Staubli VAL3: page_home_set.pjx

--- page_home_set.pjx ---
Parameters version=s7.6.3 stackSize=5000 millimeterUnit=true
Program file=alreadyExist.pgx
Program file=buildList.pgx
Program file=dataListAdd.pgx
Program file=deleteItem.pgx
Program file=listAdd.pgx
Program file=loadPage.pgx
Program file=main.pgx
Program file=markListAdd.pgx
Program file=markTraj.pgx
Program file=onEnterEvent.pgx
Program file=onExit.pgx
Program file=onF1Event.pgx
Program file=onF2Event.pgx
Program file=onF3Event.pgx
Program file=onF4Event.pgx
Program file=onF5Event.pgx
Program file=onF6Event.pgx
Program file=onF7Event.pgx
Program file=onF8Event.pgx
Program file=onLeftEvent.pgx
Program file=onRightEvent.pgx
Program file=onStart.pgx
Program file=refresh.pgx
Program file=refreshDynamic.pgx
Program file=refreshStatic.pgx
Program file=Wizard_bigBox.pgx
Program file=Wizard_smlBox.pgx
Data file=page_home_set.dtx
Library alias=page path=Disk://kernel/template/page/page.pjx
Library alias=use path=Disk://goHome/userPage/userPage.pjx
Library alias=home path=Disk://goHome/goHome.pjx
Library alias=save path=Disk://goHome/saveHomeBox/saveHomeBox.pjx
Library alias=set path=Disk://goHome/goHome.pjx
Library alias=language2 path=Disk://goHome/language/language.pjx
Library alias=cycleStatus path=Disk://cycleStatus/cycleStatus.pjx
Library alias=saveData path=Disk://saveData/saveData.pjx
Library alias=language path=Disk://kernel/language/language.pjx
Library alias=TRAJ path=Disk://trajectory/TRAJ/TRAJ.pjx
Library alias=JPOINT path=Disk://trajectory/JPOINT/JPOINT.pjx

--- page_home_set.dtx ---
public string sItems
num nKey
num nIndex
public string sEvent
num nView
num nSelected
string sList
public string sMenuUser[8]
num nRefresh
num nTime = 0.5
string sMenu
bool bLarge
bool bButton[8]
num nInsert
string sMarkList
string sDataList
num nSelected1

--- main.pgx ---
public program main()
  local num i
  local bool l_bSave
  local string sButton[3]
  local string sItems[2]
begin
  call onStart()
  do
    call refresh()
    nKey=getKey()
    call use:listevent(nKey,nIndex,sEvent)
    nView=use:nView
    nSelected=nIndex
    //
    // OVERRIDE NORMAL FUNCTIONALITY-> POLYMORPHISM
    //
    switch nKey
      case 264
        // left
        call onLeftEvent()
      break
      case 268
        // right
        call onRightEvent()
      break
      case 271
        // test
        call onF1Event()
      break
      case 272
        //
        call onF2Event()
      break
      case 273
        call onF3Event()
      break
      case 274
        call onF4Event()
      break
      case 275
        //
        call onF5Event()
      break
      case 276
        // set type
        call onF6Event()
      break
      case 277
        // DELETE
        call onF7Event()
      break
      case 278
        // NEW
        call onF8Event()
        l_bSave=true
      break
      case 270
        call onEnterEvent()
      break
    endSwitch
    // release the resource
    delay(0)
  until nKey==255 and isKeyPressed(289)==false
  // exit
  call onExit(l_bSave)
end

--- alreadyExist.pgx ---
program alreadyExist(string& x_sName[], bool& x_bUndo[])
  local num l_nX
  local num l_nY
  local string l_sString
begin
  // look if the trajectory already exist
  l_nX=40-use:nBottomX-1
  l_nY=use:nBottomY+1
  call language:message(l_sString,21)
  call use:type(l_nX,l_nY,l_sString)
  // read the new trajectory
  call use:read(l_nX+len(l_sString),l_nY,x_sName,10,false)
  if !use:bUseEscape
    call set:find(x_sName,x_bUndo)
    if x_bUndo
      call language:message(x_sName,-2)
      popUpMsg(x_sName)
    endIf
  else
    x_bUndo=true
  endIf
end

--- buildList.pgx ---
program buildList()
  local num i
  local bool l_bFound
  local num l_nCount
  local num l_nSize
  local string l_sEmpty
  local string l_sEvent
begin
  // INIT the list
  l_sEmpty=""
  call use:stringCopy(l_sEmpty,sList)
  // Build the list
  call home:getBoxSize(save:nBoxType,l_nSize)
  for i=0 to l_nSize-1
    call set:getEvent(l_sEvent,i,save:nBoxType)
    if l_sEvent!=""
      //
      // use the filter ?
      //
      // check if the bProcessList filter is active
      //
      l_bFound=true
      // update the selected item
      if l_sEvent==sEvent
        nSelected=l_nCount
      endIf
      // add
      if l_bFound
        call listAdd(l_sEvent)
        l_nCount=l_nCount+1
      endIf
    endIf
  endFor
  // update
  use:bUseRefresh=true
end

--- dataListAdd.pgx ---
program dataListAdd(string x_sEvent)
begin
  // add in the queue
  if sDataList!=""
    insert(sDataList[size(sDataList)])
  endIf
  sDataList[size(sDataList)-1]=x_sEvent
end

--- deleteItem.pgx ---
program deleteItem(bool& x_bResult)
  local string l_sMessage
  local string l_sButton[2]
  local string l_sTitle
  local bool l_bYes
begin
  x_bResult=false
  //delete it
  call language2:message(l_sMessage,3)
  call language:getYesNo(l_sButton)
  call set:getListTitle(l_sTitle)
  call use:yes_no(l_sMessage+"#"+l_sTitle+" "+sEvent,l_sButton,l_bYes)
  x_bResult=l_bYes
end

--- loadPage.pgx ---
program loadPage(string x_sPage (dimensions=1), string& x_sItems[] (dimensions=1))
// load the next page
  local num i
begin
  // look if the page libload is correct
  i=page:libLoad(x_sPage)
  if i!=0
    logMsg("[VALPLAST] INTERFACE:PAGE LIBLOAD "+x_sPage+" result "+toString("",i))
    popUpMsg("Loading page "+x_sPage+" error CODE "+toString("",i))
  else
    // copy all the field from x_sItems to the next page
    page:sItems=x_sItems
    call page:main()
    // to give back
    x_sItems=page:sItems
  endIf
end

--- markListAdd.pgx ---
program markListAdd(string x_sEvent)
begin
  // add in the queue
  if sMarkList!=""
    insert(sMarkList[size(sMarkList)])
  endIf
  sMarkList[size(sMarkList)-1]=x_sEvent
end

--- markTraj.pgx ---
program markTraj(num& x_nResult)
  local string l_sMessage[2]
  local num l_nTRAJ
  local num l_nJPOINT
  local string l_sKey
  local num i
  local string l_sItem
  local bool l_bRefresh
  local string l_sEmpty
  local num l_nView
  local string l_sEvent
  local bool l_bFound
  local num l_nCount
  local bool l_bSelected
  local num l_nSelected
  local bool l_bOk
begin
  //********************get data list*********//
  call use:stringCopy(l_sEmpty,sDataList)
  call TRAJ:getSize(l_nTRAJ)
  call JPOINT:getSize(l_nJPOINT)
  for i=0 to l_nTRAJ-1
    call TRAJ:get(l_sKey,i)
    l_sMessage="TRAJ "+l_sKey
    call dataListAdd(l_sMessage)
  endFor
  for i=0 to l_nJPOINT-1
    call JPOINT:get(l_sKey,i)
    l_sMessage="JPOINT "+l_sKey
    call dataListAdd(l_sMessage)
  endFor
  l_bRefresh=true
  do
    //******************************************//
    //******************bulid list*****************//
    for i=0 to size(sDataList)-1
      l_sEvent=sDataList[i]
      if l_sEvent!=""
        l_bFound=true
        // update the selected item
        if l_sEvent==sEvent
          nSelected=l_nCount
        endIf
        // add
        if l_bFound
          l_nCount=l_nCount+1
        endIf
      endIf
    endFor
    do

      if l_bRefresh==true
        l_bRefresh=false
        cls()
        // define your list size for default
        call use:setSizeList(0,0,22,11)
        call use:setView(false)
        call use:listcreate("")
        call use:listadd(sDataList)
        call use:clear(0,13)
        call language2:message(l_sMessage,5)
        call use:type(1,13,l_sMessage)
        call use:type(32,13,"#")
        call use:type(37,13,"OK")
        // refresh the list
        call use:selectNewField(nSelected,nIndex,nView)
        call refreshDynamic()
      else
        // refresh the Dynamic message
        if abs(clock()-nRefresh)>nTime
          call refreshDynamic()
        endIf
      endIf
      nKey=getKey()
      call use:listevent(nKey,nIndex,sEvent)
      nView=use:nView
      nSelected=nIndex
      switch nKey
        case 277
          if sEvent !=""
            if left(sDataList[nIndex],1)!="#"
              sDataList[nIndex]="# "+sDataList[nIndex]
              l_bRefresh=true
            else
              sDataList[nIndex]=right(sDataList[nIndex],len(sDataList[nIndex])-2)
              l_bRefresh=true
            endIf
          endIf
          call use:nullKey(nKey)
        break
        case 278
          l_bSelected=true
          call use:nullKey(nKey)
        break
      endSwitch
      delay(0)
    until nKey==255  or l_bRefresh==true or l_bSelected==true
    if l_bSelected==true
      //**********************已经选择的部分**********************//
      call use:stringCopy(l_sEmpty,sMarkList)
      do
        l_bRefresh=false
        cls()
        // create the list
        call use:setSizeList(12,0,25,11)
        call use:clear(0,13)
        call language2:message(l_sMessage,8)
        call use:type(31,13,l_sMessage)
        call language2:message(l_sMessage,7)
        call use:type(36,13,l_sMessage)
        // get the value

        //add mark list
        for i=0 to size(sDataList)-1
          if left(sDataList[i],1)=="#"
            call markListAdd(right(sDataList[i],len(sDataList[i])-2))
          endIf
        endFor
        if sMarkList==""
          l_nSelected=0
        else
          l_nSelected=size(sMarkList)
        endIf
        call language2:message(l_sMessage[0],52)
        call language2:message(l_sMessage[1],53)

        call use:listcreate(l_sMessage[0]+toString("",l_nSelected)+l_sMessage[1])
        //
        for i=0 to size(sMarkList)-1
          l_sItem=sMarkList[i]
          call use:listadd(l_sItem)
        endFor

        //////////bulid list
        ////////////////////
        // list update
        call use:listupdate(min(nInsert,size(sMarkList)))

        // Select ???
        do
          nKey=get()
          call use:listevent(nKey,nInsert,l_sItem)
          // release the resource
          if nKey==277
            l_bRefresh=true
            l_bSelected=false
            call use:nullKey(nKey)
          endIf
          if nKey==278
            if sMarkList==""
              call language2:message(l_sMessage,9)
              popUpMsg(l_sMessage)
              cls()
              use:bUseRefresh=true
              wait(getKey( )==-1)
              x_nResult=-1
              return
            endIf
            call set:IsUseSameTool(sMarkList,l_bOk)
            if l_bOk==false
              call language2:message(l_sMessage,54)
              popUpMsg(l_sMessage)
              cls()
              use:bUseRefresh=true
               wait(getKey( )==-1)
              x_nResult=-1
              return
            endIf
            cls()
            use:bUseRefresh=true
            x_nResult=0
            call use:nullKey(nKey)
            return
          endIf
        until nKey==255 or l_bRefresh
        delay(0)
      until nKey==255 or l_bRefresh
      //*****************************************************************//
    endIf
  until nKey==255
  if nKey==255
    x_nResult=-1
  endIf
  // update
  call use:nullKey(nKey)
  use:bUseRefresh=true
  //*******************************************//

end

--- onEnterEvent.pgx ---
program onEnterEvent()
  local num l_nResult
  local string l_sMessage
begin
  if sEvent!=""

    if  save:nBoxType==1
      set:bWizard=false
      call set:editSmlData(sEvent,l_nResult)
      call language2:message(l_sMessage,4)
      call use:timerDialog(l_sMessage,0)
      call set:onSave()
    elseIf save:nBoxType==2
      set:bWizard=false
      call set:editBigData(sEvent,l_nResult)
      call language2:message(l_sMessage,4)
      call use:timerDialog(l_sMessage,0)
      call set:onSave()
    endIf
  endIf
end

--- onExit.pgx ---
public program onExit(bool x_bSave)
begin
 save:libSave()
 call set:onSave()
end

--- onF1Event.pgx ---
program onF1Event()
  local bool l_NoBox
  local bool l_bStop
  local string l_sDynamicStu[3]
  local num l_n
  local string l_sMessage
begin
  // look if the bButton is enable
  if bButton[0]
    if cycleStatus:bIsHome
       call language2:message(l_sMessage,58)
       popUpMsg(l_sMessage)
      return
    endIf
    call set:_IsUseingBox(l_NoBox)
    if l_NoBox==true
           call language2:message(l_sMessage,59)
       popUpMsg(l_sMessage)
      return
    endIf
    if workingMode( )==1 and !cycleStatus:bCycle  and !cycleStatus:bIsHome and !l_NoBox
      //      call use:timerDialog("请选择夹爪号,默认为1",2)
      //      call _setToolType()
      taskCreate "GOHOME",100,set:GOHOME()
      wait(taskStatus("GOHOME")==1)
      cls()

      cycleStatus:bHoming=true
      l_sDynamicStu[0]=">"
      l_sDynamicStu[1]=">>"
      l_sDynamicStu[2]=">>>"
      set:sHomingStatus=""
      do
        // set the menu
        //call use:setMenu(sMenu,true,-1)
        call use:type(32,13,"STOP ")
        nKey=getKey()
        // REFRESH
        if nKey==277
          stopMove()
          taskKill("GOHOME")
          wait(taskStatus("GOHOME")==-1)
          resetMotion( )
          l_bStop=true
        endIf
          call language2:message(l_sMessage,60)
        call use:timerDialog(l_sMessage+l_sDynamicStu[l_n]+"#"+set:sHomingStatus,0.5)
        if l_n==2
          l_n=0
        else
          l_n=l_n+1
        endIf
        delay(0.3)
      until l_bStop or  cycleStatus:bHoming==false  or cycleStatus:bIsHome
      cycleStatus:bHoming=false
      use:bUseRefresh =true
      cls()
    endIf
  endIf
end

--- onF2Event.pgx ---
program onF2Event()
begin
end

--- onF3Event.pgx ---
program onF3Event()
begin
end

--- onF4Event.pgx ---
public program onF4Event()
begin
end

--- onF5Event.pgx ---
program onF5Event()
begin
end

--- onF6Event.pgx ---
program onF6Event()
  local string l_sItem
begin
  //设定对话框位置及尺寸大小
  call use:setSizeList(15,9,15,2)
  //建立对话款
  call language2:message(l_sItem,61)
  call use:listcreate(l_sItem)
  //增加一栏数据
   call language2:message(l_sItem,1)
  call use:listadd(l_sItem)
  //再增加一栏数据
   call language2:message(l_sItem,2)
  call use:listadd(l_sItem)
  //更新光标选择位置
    call use:listupdate(0)
  //设置循环直至按ESC推出
  do
    nKey=get()
    call use:listevent(nKey,nIndex,sEvent)
    if nKey==270
      if nIndex==0
        save:nBoxType=1
      else
        save:nBoxType=2
      endIf
    endIf
  until nKey==255 or nKey==270
  call use:nullKey(nKey)
  call buildList()
  cls()
  use:bUseRefresh=true

end

--- onF7Event.pgx ---
program onF7Event()
  local bool l_bYes
  local num l_nResult
  local string l_sMessage
begin
  if bButton[6] and sEvent!=""
    call deleteItem(l_bYes)
    if l_bYes
      call set:delete(sEvent,l_nResult)
      if l_nResult==0
        logMsg("[KERNEL] INTERFACE:Delete the box: "+" "+sEvent)
        call language2:message(l_sMessage,4)
        call use:timerDialog(l_sMessage,0)
        call set:onSave()
        call buildList()
      else
        popUpMsg("error code: "+toString("",l_nResult))
      endIf
    endIf
    call use:nullKey(nKey)
  endIf
end

--- onF8Event.pgx ---
program onF8Event()
  local bool l_bUndo
  local num l_nResult
  local string l_sNew
  local string l_sMessage
begin
  if bButton[7]
    // new one
    call alreadyExist(l_sNew,l_bUndo)
    if !l_bUndo and l_sNew!=""
      call set:new(l_sNew,l_nResult)
      if l_nResult==0
          set:bWizard=true
        if save:nBoxType==1
          call Wizard_smlBox(l_sNew,l_nResult)
        elseIf save:nBoxType==2
          call set:editBigData(l_sNew,l_nResult)
        endIf
        ///////////////////////////////////
        if l_nResult==0
          call language2:message(l_sMessage,4)
          call use:timerDialog(l_sMessage,0)
          call set:onSave()
          sEvent=l_sNew
          call buildList()
        else
           call set:delete(l_sNew,l_nResult)
           call set:onSave()
       endIf
      endIf
    endIf
  endIf
end

--- onLeftEvent.pgx ---
program onLeftEvent()
begin
  call save:BackBoxType()
  call buildList()
end

--- onRightEvent.pgx ---
program onRightEvent()
begin
  call save:FwdBoxType()
  call buildList()
end

--- onStart.pgx ---
program onStart()
begin
  call language2:setLanguage(language2:libPath()+"/"+saveData:language)
  if save:nBoxType<1 or save:nBoxType>2
    save:nBoxType=1
  endIf
  // reset the Key pressure
  call use:nullKey(nKey)
  //bulidList
  call buildList()
end

--- refresh.pgx ---
program refresh()
begin
  if (nKey>=270 and nKey<=278) or use:bUseRefresh
    call refreshStatic()
    call refreshDynamic()
  else
    // refresh the Dynamic message
    if abs(clock()-nRefresh)>nTime
      call refreshDynamic()
    endIf
  endIf
end

--- refreshDynamic.pgx ---
program refreshDynamic()
begin
  // DO NOT CHANGE
  nRefresh=clock()
  use:bUseRefresh=false
  //
end

--- refreshStatic.pgx ---
program refreshStatic()
  local string l_sMessage
begin
  cls()
  //
  // set the view of the page..
  //
  // SET THE PAGE NUMBER
  use:nPage=300
  // USE <>PROFILE for <>PAGE
  if cycleStatus:bCycle
    use:nPage=301
  endIf

  // load the menu page
  // SET THE VIEW OF THE PAGE
  call language2:page(l_sMessage,use:nPage)
  // define the menu
  call use:stringToArray(l_sMessage,sMenu)
  // set the menu
  call use:setMenu(sMenu,true,3)
  call use:getMenu(sMenu,bButton)
  //
  // CREATE THE LIST
  //
  // define your list size for default
  call use:setSizeList(16,0,22,11)
  call use:setView(bLarge)

  call set:getListTitle(l_sMessage)
  call use:listcreate(l_sMessage)
  //
  call use:listadd(sList)
  //
  // refresh the list
  call use:selectNewField(nSelected,nIndex,nView)
  //

end

--- Wizard_bigBox.pgx ---
program Wizard_bigBox()
begin
end

--- Wizard_smlBox.pgx ---
program Wizard_smlBox(string x_sName, num& x_nResult)
begin
  if set:bWizard
    call markTraj(x_nResult)
  endIf
  if x_nResult==0
    if set:bWizard
      call set:loadMarkData(x_sName,sMarkList)
    endIf
    if x_nResult==0
      call set:editSmlData(x_sName,x_nResult)
      if x_nResult==0
        call set:onSave()
      endIf
    endIf
  endIf

end
